// TIA Portal V18 export
DATA_BLOCK "delete2"   // DB59
VERSION : 0.1
// stored: AutoNumber true, DBAccessibleFromOPCUA true, InstanceOfName _ML2_target_supplier, InstanceOfType FB
"_ML2_target_supplier"
   // VAR_INPUT
   //    ALLOWED : Bool := TRUE;
   //    xServiceKey : Bool := FALSE;
   //    xManButtonAny : Bool := FALSE;
   //    xSwAutoCycle : Bool := FALSE;
   //    xXrayCycleRuning : Bool;
   //    xGoToNextDefect : Bool := FALSE;
   //    xGoToPrevDefect : Bool := FALSE;
   //    xHome : Bool;
   //    xLoad : Bool;
   //    xControl1 : Bool;
   //    xControl2 : Bool;
   //    xDefectSave : Bool := FALSE;
   //    xDefectsReset : Bool := FALSE;
   //    Spots_pos_AR : "typeSpotList";
   //    CurPositios : "typePositions";
   //    ACK : Bool;
   //    ArrivedAll : Bool;
   //    HomePos : "typePositions";
   //    LoadPos : "typePositions";
   //    Control1Pos : "typePositions";
   //    Control2Pos : "typePositions";
   //    bSoftStop : Bool;
   // END_VAR
   // VAR_OUTPUT
   //    ExecuteAllAxisTogether : Bool;
   //    mdNotAllowed : Bool := FALSE;
   //    mdServiceKey : Bool := FALSE;
   //    mdCycle : Bool := FALSE;
   //    mdSemi : Bool := FALSE;
   //    mdMan : Bool := TRUE;
   //    wsMODE : WString := WSTRING#'Ручной';
   //    wsTarget : WString := WSTRING#'цель не задана';
   //    er_ws : WString;
   // END_VAR
   // VAR_IN_OUT
   //    Target_pos : "typePositions";
   //    DefectsDB : "typeDefectsDB";
   //    hmiGoToDefect : Bool := FALSE;
   //    hmiGotoSpot : Bool := FALSE;
   //    SPOT_i : Int := 0;
   //    xyBeepDoneDefects : Bool := FALSE;
   // END_VAR
   // VAR
   //    def_util_db { S7_SetPoint := 'True'} : "defects_util";
   //    mdSemi_was : Bool := FALSE;
   //    st_goToDefectNow : Bool;
   //    q0_auto : Bool;
   //    q00_semi : Bool;
   //    q1_spot : Bool;
   //    p1_spot : Bool;
   //    q2_defect : Bool;
   //    p2_defect : Bool;
   //    q99_none : Bool;
   //    q_auto_waiting : Bool;
   //    block1 { S7_SetPoint := 'True'} : "_ML2_ts_block1";
   //    p3_home : Bool;
   //    q3_home : Bool;
   //    p4_load : Bool;
   //    q4_load : Bool;
   //    p5_control1 : Bool;
   //    q5_control1 : Bool;
   //    p6_control2 : Bool;
   //    q6_control2 : Bool;
   // END_VAR
BEGIN
   Spots_pos_AR.N := 4;
   Spots_pos_AR.pos_AR[1].M1Z := 11.0;
   Spots_pos_AR.pos_AR[2].M1Z := 33.0;
   Spots_pos_AR.pos_AR[3].M1Z := 55.0;
   Spots_pos_AR.pos_AR[4].M1Z := 44.0;
   Spots_pos_AR.pos_AR[5..30].M1Z := 0.0;
   Spots_pos_AR.pos_AR[1..30].M2Y := 0.0;
   Spots_pos_AR.pos_AR[1..30].M3X := 0.0;
   Spots_pos_AR.pos_AR[1..30].M4O1 := 0.0;
   Spots_pos_AR.pos_AR[1..30].M5O2 := 0.0;
   CurPositios.M1Z := 0.0;
   CurPositios.M2Y := 0.0;
   CurPositios.M3X := 0.0;
   CurPositios.M4O1 := 0.0;
   CurPositios.M5O2 := 0.0;
   def_util_db.xBdefect_inc := FALSE;
   def_util_db.xBdefect_dec := FALSE;
   def_util_db.xDefectsClearAll := FALSE;
   def_util_db.xDefect_Save := FALSE;
   def_util_db.positions.M1Z := 0.0;
   def_util_db.positions.M2Y := 0.0;
   def_util_db.positions.M3X := 0.0;
   def_util_db.positions.M4O1 := 0.0;
   def_util_db.positions.M5O2 := 0.0;
   def_util_db.go_to_defect_now := FALSE;
   def_util_db.xyBeepDone := FALSE;
   def_util_db.mem1 := FALSE;
   def_util_db.mem2 := FALSE;
   def_util_db.xdefect_dec_was := FALSE;
   def_util_db.xdefect_inc_was := FALSE;
   def_util_db.xDefect_Save_was := FALSE;
   def_util_db.xDefectsClearAll_was := FALSE;
END_DATA_BLOCK
